FUNCTION_BLOCK PUBLIC PIZZA_OVEN
VAR_INPUT

	Pizza_in 	: 		BOOL:=FALSE;
	Pizza_out 	:		BOOL:=FALSE;

	fbTrig		: 	R_TRIG;
	fbTrig2		: 	R_TRIG;
END_VAR
VAR_OUTPUT
	PizzaStatus	: 	STRING;
END_VAR
VAR
	fbTimer		: 	TON;
	PizzaInOven	: 	BOOL;
	PizzaOnDeck	: 	BOOL;
	PizzaDone	: 	BOOL;
 	
	iState		:  	DINT:=0;
	bBurned:		BOOL;
END_VAR


//control buttons
		fbTrig(CLK:=Pizza_in);//load pizza button clicked trggered
IF		fbTrig.Q THEN		//When Triggerd 
		PizzaOnDeck:=TRUE;	
		//Pizza_in:=FALSE;
		//fbTrig(clk:=FALSE);
END_IF		

	fbTrig2(CLK:=Pizza_out); 
IF 	Pizza_out THEN
	PizzaDone:=FALSE;
	//Pizza_out:=FALSE;
		//fbTrig2(clk:=Pizza_out);
END_IF


//status changes
CASE iState OF 
0:	IF PizzaOnDeck AND NOT PizzaInOven THEN
		PizzaOnDeck:=FALSE;
		PizzaInOven:=TRUE;
		iState:=10;
	END_IF
10:	PizzaStatus:='cooking...';
IF PizzaInOven THEN
fbTimer(IN:=PizzaInOven,PT:=T#3S);
	END_IF
IF fbTimer.Q THEN
	//PizzaInOven:=FALSE;
	
	iState:=20;
	
END_IF
	
20:	//Pizza out.
	
	IF  NOT PizzaDone THEN

	PizzaInOven:=FALSE;
	PizzaDone:=TRUE;
	fbTimer(IN:=FALSE);
	iState:=0;
	ELSE 
		bBurned:=TRUE;
	END_IF
	
END_CASE

PROPERTY Burned : BOOL;
GET
bBurned:=Burned;
END_GET
SET
Burned:=bBurned;
END_SET
END_PROPERTY

METHOD PUBLIC MethodPizza : UDINT
VAR_INPUT
burned 		:BOOL;
	bBurned			: BOOL;
END_VAR
VAR

END_VAR
IF burned THEN
	
	bBurned:=TRUE;
END_IF
END_METHOD

END_FUNCTION_BLOCK

(* stored: Version 1.1.0.1, ProductVersion 3.1.4022.6
   POU PIZZA_OVEN: Id {e54d8141-8c6a-4975-af63-b1ccd7a5bba4}, SpecialFunc None
   Property Burned: Id {1d1409a6-25fd-400a-bee1-b98e880d4431}
   Get Get: Id {0cd453c2-a84f-4940-8569-6ea5216b1c29}
   Set Set: Id {7fa32c2c-01e8-4699-bd9b-b92865c765e7}
   Method MethodPizza: Id {973a8685-4554-4338-ac21-4d340b906904} *)
